// Block: PPrgArchive1

DATA_BLOCK PPrgArchive1
VERSION : 0.1
   NON_RETAIN
   VAR
      PRG : Array[1..100] of PPrg_Data;
   END_VAR

BEGIN
   // No initialization required
END_DATA_BLOCK
